FUNCTION_BLOCK FB_PumpBACnet2 IMPLEMENTS I_Pump
VAR_INPUT CONSTANT
	fbClient : FB_BACnet_Client;
END_VAR
VAR_OUTPUT
END_VAR
VAR
	//Properties
	eControlMode : E_PumpControlMode := E_PumpControlMode.OFF;
	bError : BOOL;
	bOperating : BOOL;
	fPowerRating : REAL;
	fPressure : REAL;
	bSetOn : BOOL := FALSE;
	fSetpoint : REAL := 0;
	fSpeed : REAL;
	fVolumeFlow : REAL;	

	//BACnet parameters
	nPriority : BYTE := 12;
	
	//BACnet Mapping
	ContModeBAC		:	FB_BACnetRM_MO := (Client := fbClient, nObjectInstance :=0);		//Pump Control mode (speed, var/const pressure)
	ErrorBAC		:	FB_BACnetRM_BI := (Client := fbClient, nObjectInstance :=13);		//Error
	OperatingBAC	:	FB_BACnetRM_BI := (Client := fbClient, nObjectInstance :=10);		//Operation active/inactive
	PowerRatingBAC	:	FB_BACnetRM_AI := (Client := fbClient, nObjectInstance :=4);		//Current power
	PressureBAC		:	FB_BACnetRM_AI := (Client := fbClient, nObjectInstance :=3);		//Estimated pressure difference
	SetpointBAC		:	FB_BACnetRM_AO := (Client := fbClient, nObjectInstance :=0);		//Setpoint
	SetOnBAC		:	FB_BACnetRM_BO := (Client := fbClient, nObjectInstance :=0);		//Turn on/off
	SpeedBAC		:	FB_BACnetRM_AI := (Client := fbClient, nObjectInstance :=1);		//Estimated speed
	VolumeFlowBAC	:	FB_BACnetRM_AI := (Client := fbClient, nObjectInstance :=2);		//Estimated volume flow

END_VAR

PROPERTY ControlMode : E_PumpControlMode
GET
ControlMode := THIS^.eControlMode;
END_GET
SET
THIS^.eControlMode := ControlMode;
END_SET
END_PROPERTY

PROPERTY Error : BOOL
GET
Error := THIS^.bError;
END_GET
SET
THIS^.bError := Error;
END_SET
END_PROPERTY

PROPERTY Operating : BOOL
GET
Operating := THIS^.bOperating;
END_GET
SET
THIS^.bOperating := Operating;
END_SET
END_PROPERTY

PROPERTY PowerRating : REAL
GET
PowerRating := THIS^.fPowerRating;
END_GET
SET
THIS^.fPowerRating := PowerRating;
END_SET
END_PROPERTY

PROPERTY Pressure : REAL
GET
Pressure := THIS^.fPressure;
END_GET
SET
THIS^.fPressure := Pressure;
END_SET
END_PROPERTY

METHOD Run
//Run BACnet Client
(*fbClient();

//Read BACnet values
ErrorBAC(bPresentValue=>bError);
OperatingBAC(bPresentValue=>bOperating);
PowerRatingBAC(fPresentValue=>fPowerRating);
PressureBAC(fPresentValue=>fPressure);
SpeedBAC(fPresentValue=>fSpeed);
VolumeFlowBAC(fPresentValue=>fVolumeFlow);

//Write BACnet values
//Set pump values depending on defined ControlMode
IF eControlMode = E_PumpControlMode.OFF THEN
	//Set pump to off
	SetOnBAC(bPv:=FALSE,bEnablePv:=TRUE,ePriority:=nPriority);
	ContModeBAC(nPv:=eControlMode,bEnablePv:=TRUE,ePriority:=nPriority);
	SetpointBAC(fPv:=0,bEnablePv:=TRUE,ePriority:=nPriority);
ELSIF eControlMode = E_PumpControlMode.NONE THEN
	//Release
	SetOnBAC(bNullPv:=TRUE,ePriority:=nPriority); 	//Clear entry
	ContModeBAC(bNullPv:=TRUE,ePriority:=nPriority); //Clear entry
	SetpointBAC(bNullPv:=TRUE,ePriority:=nPriority); //Clear entry
ELSE
	//Set pump to on and set setpoint
	SetOnBAC(bPV:=TRUE,bEnablePv:=TRUE,ePriority:=nPriority);
	ContModeBAC(nPV:=eControlMode,bEnablePv:=TRUE,ePriority:=nPriority);
	SetpointBAC(fPV:=fSetpoint,bEnablePv:=TRUE,ePriority:=nPriority);
END_IF

*)
END_METHOD

PROPERTY SetOn : BOOL
GET
SetOn := THIS^.bSetOn;
END_GET
SET
THIS^.bSetOn := SetOn;
END_SET
END_PROPERTY

PROPERTY Setpoint : REAL
GET
Setpoint := THIS^.fSetpoint;
END_GET
SET
THIS^.fSetpoint := Setpoint;
END_SET
END_PROPERTY

PROPERTY Speed : REAL
GET
Speed := THIS^.fSpeed;
END_GET
SET
THIS^.fSpeed := Speed;
END_SET
END_PROPERTY

PROPERTY VolumeFlow : REAL
GET
VolumeFlow := THIS^.fVolumeFlow;
END_GET
SET
THIS^.fVolumeFlow := VolumeFlow;
END_SET
END_PROPERTY

END_FUNCTION_BLOCK

(* stored: Version 1.1.0.1, ProductVersion 3.1.4024.3
   POU FB_PumpBACnet2: Id {165c6dd0-ac9a-42e2-8614-3ed8dafaefcb}, SpecialFunc None
   Property ControlMode: Id {5c3b4501-6c3e-4417-b93b-fd3c7ff3ea59}
   Get Get: Id {e302f8c0-109c-4c40-851f-660acf7b9cad}
   Set Set: Id {9d554b36-8089-4c0b-8b9d-64d4ce524955}
   Property Error: Id {e5122c8e-94ab-4cba-ae19-ae45af740a89}
   Get Get: Id {cc535b96-e743-423e-b470-607a2f3049cc}
   Set Set: Id {6458b08e-0e8c-4e48-a1d6-12dfeffb0857}
   Property Operating: Id {4dc4cd74-ff44-4c4d-ae00-0059778e3b78}
   Get Get: Id {9d18471a-002f-4da4-bdb9-a2ff14fd88ea}
   Set Set: Id {76eed797-f462-4cc4-8ee7-189919e0df46}
   Property PowerRating: Id {fd9c959a-95fc-4efa-bf87-37672456dc97}
   Get Get: Id {7cc7fa91-301e-458a-8eae-fb4b54c237bb}
   Set Set: Id {e2fa6912-5b3c-43b8-a28f-cd65a1f5169e}
   Property Pressure: Id {2f49c6af-8df9-4a62-a963-9bc0e13a5e56}
   Get Get: Id {2dc70fd3-df75-4433-9ff8-17f4ea0196c6}
   Set Set: Id {6e692c93-cc69-406b-a9b0-4b53b0568d4a}
   Method Run: Id {28d90e17-304c-4e46-b3c3-3ac8fce7188c}
   Property SetOn: Id {01a277b9-2e24-41b1-8ccd-9da4fa529386}
   Get Get: Id {4e844d26-9fae-486c-9cb3-2d7d92db1f75}
   Set Set: Id {42046a70-5cf9-4c45-ad02-f660564abfdd}
   Property Setpoint: Id {5f5aac7c-29c2-43fd-bc1e-5660741af6e4}
   Get Get: Id {9ac4a73d-c19f-4730-b934-7926dc5c2380}
   Set Set: Id {5274a693-3a8d-415a-bdcd-a16f9d7fc971}
   Property Speed: Id {ebe85331-e5bb-45bb-b572-320627f2bf26}
   Get Get: Id {5c3a3e93-c9f8-42ea-904a-7168b79f5ccc}
   Set Set: Id {43a3fcf9-5680-4333-bd26-91c9a1baebab}
   Property VolumeFlow: Id {ac0e2c43-67a7-493d-b60d-ad1224890df9}
   Get Get: Id {4a44909c-da5f-4859-8d1d-8771c6c92698}
   Set Set: Id {9cb5baa2-dbf1-4b5c-8af5-31d6839add17} *)
